INTERFACE I_Queue EXTENDS I_Collection, I_EventEmitter

METHOD PUBLIC Enqueue
VAR_INPUT
	Item : ANY;
END_VAR
END_METHOD

METHOD PUBLIC TryDequeue : BOOL;
VAR_INPUT
	Destination : ANY;
END_VAR
END_METHOD

METHOD PUBLIC TryPeek : BOOL;
VAR_INPUT
	Destination : ANY;
END_VAR
END_METHOD

END_INTERFACE

(* stored: Version 1.1.0.1, ProductVersion 3.1.4024.12
   Itf I_Queue: Id {9ef9041f-cd02-4017-af5b-d6ee42f4947a}
   Method Enqueue: Id {a8efe73a-c86f-4d9c-81d8-371b69901091}
   Method TryDequeue: Id {3417b1ed-3e3a-4043-ad29-b14a057c5ec8}
   Method TryPeek: Id {60f460c4-d3b6-43db-96bb-95be3f404eb6} *)
